FUNCTION_BLOCK FB_NormallyOpenSensor IMPLEMENTS I_Sensor
VAR
	Input AT %I* : BOOL;
END_VAR

PROPERTY IsActive : BOOL
GET
IsActive := Input;
END_GET
END_PROPERTY

END_FUNCTION_BLOCK

(* stored: Version 1.1.0.1, ProductVersion 3.1.4024.9
   POU FB_NormallyOpenSensor: Id {62763c25-bf0a-4cc0-9276-55059e992b67}, SpecialFunc None
   Property IsActive: Id {55032022-ddfe-4e69-8bf0-bd902a6ee556}
   Get Get: Id {f05c2218-f255-4b80-aa34-6ec6c6918596} *)
